FUNCTION TryConvert_USINT_TO_LINT : BOOL
VAR_INPUT
	in : USINT;
	out : REFERENCE TO LINT;
END_VAR

out := USINT_TO_LINT(in);
TryConvert_USINT_TO_LINT := TRUE;

END_FUNCTION

(* stored: Version 1.1.0.1, ProductVersion 3.1.4024.12
   POU TryConvert_USINT_TO_LINT: Id {54f04683-ec08-48f1-8192-b2a1124bc132}, SpecialFunc None *)
